(* Logix 5000 project; controller BreakGroup_US vendor 1 type 14 code 211 rev 32.16; software revision 32.05; part 3 of 8 *)
(* tags used below, declared in another part *)
   Emg_Stop : BOOL;
   Gantry_2_Horizontal_Start : BOOL;
   Gantry_2_Tilter_LH_Start : BOOL;
   Gantry_2_Tilter_RH_Start : BOOL;
   Gantry_2_vertical_Start : BOOL;
   HMI_Gantry_02_Hor_PB : SINT;
   HMI_Gantry_2_Tilter_LH_PB : SINT;
   HMI_Gantry_2_Tilter_RH_PB : SINT;
   HMI_Gantry_2_vertical_PB : SINT;
   HMI_MAN_GTY2_HORI_STOP : BOOL;
   HMI_MAN_GTY2_TIL2_STOP : BOOL;
   HMI_MAN_GTY2_VERT_STOP : BOOL;
   MAN_GTY2_HORI_HOME : TIMER;
   MAN_GTY2_TIL1_HOME : TIMER;
   MAN_GTY2_TIL2_HOME : TIMER;
   MAN_GTY2_VERT_HOME : TIMER;
   RCP_GY_02_Horizontal : RCP_Servo_02;
   RCP_GY_02_Vertical : RCP_Servo_02;
   RCP_Tilt_Axis_Master : RCP_Servo_02;
   RCP_Tilt_Axis_Slave : RCP_Servo_02;
   ST10_Trolley1Lock_Cyl_01_Extended : ALIAS FOR MCP_PT01:1:I.0;
   ST10_Trolley1LockCyl_01_Retracted : ALIAS FOR MCP_PT01:1:I.1;
   ST10_Trolley_Present_Sensor : ALIAS FOR MCP_PT01:1:I.2;
   ST10_TrolleyTopSideProductPresentSensor : ALIAS FOR MCP_PT01:1:I.3;
   ST20_Trolley_Present_Sensor_02 : ALIAS FOR MCP_PT01:1:I.6;
   ST20_TrolleyTopSideProductPresentSensor : ALIAS FOR MCP_PT01:4:I.3;
   ST30_Auto_SS : ALIAS FOR MCP_PT01:6:I.3;
   ST30_Emg_Push_Buttion : ALIAS FOR MCP_PT01:5:I.7;
   ST30_Home_PB : ALIAS FOR MCP_PT01:6:I.2;
   ST30_Hydro_motor : ALIAS FOR MCP_PT01:5:I.6;
   ST30_IndexingTableHomePositionSensor : ALIAS FOR MCP_PT01:4:I.5;
   ST30_IndexPlateLockCyl1Extended : ALIAS FOR MCP_PT01:4:I.6;
   ST30_IndexPlateLockCyl1Retracted : ALIAS FOR MCP_PT01:4:I.7;
   ST30_IndexPlateLockCyl2Extended : ALIAS FOR MCP_PT01:5:I.0;
   ST30_IndexPlateLockCyl2Retracted : ALIAS FOR MCP_PT01:5:I.1;
   ST30_Manual_SS : ALIAS FOR MCP_PT01:6:I.4;
   ST30_PressUnitCyl_1Extended : ALIAS FOR MCP_PT01:5:I.2;
   ST30_PressUnitCyl_1Retracted : ALIAS FOR MCP_PT01:5:I.3;
   ST30_PressUnitCyl_2Extended : ALIAS FOR MCP_PT01:5:I.4;
   ST30_PressUnitCyl_2Retracted : ALIAS FOR MCP_PT01:5:I.5;
   ST30_Product_Present_Sensor : ALIAS FOR MCP_PT01:4:I.4;
   ST30_Reset_PB : ALIAS FOR MCP_PT01:6:I.5;
   ST30_Start_PB : ALIAS FOR MCP_PT01:6:I.0;
   ST30_Stop_PB : ALIAS FOR MCP_PT01:6:I.1;
   ST40_Auto_SS : ALIAS FOR MCP_PT01:10:I.5;
   ST40_EMG_PB : ALIAS FOR MCP_PT01:10:I.1;
   ST40_Home_PB : ALIAS FOR MCP_PT01:10:I.4;
   ST40_IndexingTableHomePositionSensor : ALIAS FOR MCP_PT01:6:I.7;
   ST40_IndexPlateLockCyl01_Extended : ALIAS FOR MCP_PT01:7:I.0;
   ST40_IndexPlateLockCyl01_Retracted : ALIAS FOR MCP_PT01:7:I.1;
   ST40_IndexPlateLockCyl02_Extended : ALIAS FOR MCP_PT01:7:I.2;
   ST40_IndexPlateLockCyl02_Retracted : ALIAS FOR MCP_PT01:7:I.3;
   ST40_Manual_SS : ALIAS FOR MCP_PT01:10:I.6;
   ST40_ProductPresentSensor : ALIAS FOR MCP_PT01:6:I.6;
   ST40_Reset_PB : ALIAS FOR MCP_PT01:10:I.7;
   ST40_Start_PB : ALIAS FOR MCP_PT01:10:I.2;
   ST40_Stop_PB : ALIAS FOR MCP_PT01:10:I.3;
   ST50_Auto_SS : ALIAS FOR MCP_PT01:15:I.1;
   ST50_Conv_End_Sensor : ALIAS FOR MCP_PT01:11:I.7;
   ST50_Conv_Home_Sensor : ALIAS FOR MCP_PT01:11:I.6;
   ST50_EMG_PB : ALIAS FOR MCP_PT01:14:I.5;
   ST50_Home_PB : ALIAS FOR MCP_PT01:15:I.0;
   ST50_IndexPlateLockCyl01_Extended : ALIAS FOR MCP_PT01:11:I.2;
   ST50_IndexPlateLockCyl01_Retracted : ALIAS FOR MCP_PT01:11:I.3;
   ST50_IndexPlateLockCyl02_Extended : ALIAS FOR MCP_PT01:11:I.4;
   ST50_IndexPlateLockCyl02_Retracted : ALIAS FOR MCP_PT01:11:I.5;
   ST50_IndexTableHomePositionSensor : ALIAS FOR MCP_PT01:11:I.1;
   ST50_Manual_SS : ALIAS FOR MCP_PT01:15:I.2;
   ST50_Product_Present_Sensor : ALIAS FOR MCP_PT01:11:I.0;
   ST50_Reset_PB : ALIAS FOR MCP_PT01:15:I.3;
   ST50_Start_PB : ALIAS FOR MCP_PT01:14:I.6;
   ST50_Stop_PB : ALIAS FOR MCP_PT01:14:I.7;
   ST60_Auto_SS : ALIAS FOR MCP_PT01:20:I.2;
   ST60_Conv_End_Sensor : ALIAS FOR MCP_PT01:16:I.3;
   ST60_Conv_Home_Sensor : ALIAS FOR MCP_PT01:16:I.2;
   ST60_EMG_PB : ALIAS FOR MCP_PT01:19:I.6;
   ST60_Home_PB : ALIAS FOR MCP_PT01:20:I.1;
   ST60_Hydro_Motor : ALIAS FOR MCP_PT01:17:I.0;
   ST60_IndexPlateLockCyl01_Extended : ALIAS FOR MCP_PT01:15:I.6;
   ST60_IndexPlateLockCyl01_Retracted : ALIAS FOR MCP_PT01:15:I.7;
   ST60_IndexPlateLockCyl02_Extended : ALIAS FOR MCP_PT01:16:I.0;
   ST60_IndexPlateLockCyl02_Retracted : ALIAS FOR MCP_PT01:16:I.1;
   ST60_IndexTableHomePositionSensor : ALIAS FOR MCP_PT01:15:I.5;
   ST60_Manual_SS : ALIAS FOR MCP_PT01:20:I.3;
   ST60_Press_Unit_Cyl01_Extended : ALIAS FOR MCP_PT01:16:I.4;
   ST60_Press_Unit_Cyl01_Retracted : ALIAS FOR MCP_PT01:16:I.5;
   ST60_Press_Unit_Cyl02_Extended : ALIAS FOR MCP_PT01:16:I.6;
   ST60_Press_Unit_Cyl02_Retracted : ALIAS FOR MCP_PT01:16:I.7;
   ST60_Product_Present_Sensor : ALIAS FOR MCP_PT01:15:I.4;
   ST60_Reset_PB : ALIAS FOR MCP_PT01:20:I.4;
   ST60_Start_PB : ALIAS FOR MCP_PT01:19:I.7;
   ST60_Stop_PB : ALIAS FOR MCP_PT01:20:I.0;
   ST70_Auto_SS : ALIAS FOR MCP_PT01:22:I.1;
   ST70_Conv_End_Sensor : ALIAS FOR MCP_PT01:21:I.4;
   ST70_Conv_Home_Sensor : ALIAS FOR MCP_PT01:21:I.3;
   ST70_EMG_PB : ALIAS FOR MCP_PT01:21:I.5;
   ST70_Home_PB : ALIAS FOR MCP_PT01:22:I.0;
   ST70_IndexPlateLockCyl01_Extended : ALIAS FOR MCP_PT01:20:I.7;
   ST70_IndexPlateLockCyl01_Retracted : ALIAS FOR MCP_PT01:21:I.0;
   ST70_IndexPlateLockCyl02_Extended : ALIAS FOR MCP_PT01:21:I.1;
   ST70_IndexPlateLockCyl02_Retracted : ALIAS FOR MCP_PT01:21:I.2;
   ST70_IndexTableHomePositionSensor : ALIAS FOR MCP_PT01:20:I.6;
   ST70_Manual_SS : ALIAS FOR MCP_PT01:22:I.2;
   ST70_Product_Present_Sensor : ALIAS FOR MCP_PT01:20:I.5;
   ST70_Reset_PB : ALIAS FOR MCP_PT01:22:I.3;
   ST70_Start_PB : ALIAS FOR MCP_PT01:21:I.6;
   ST70_Stop_PB : ALIAS FOR MCP_PT01:21:I.7;
   ST_20Trolley_1LockCylExtended : ALIAS FOR MCP_PT01:1:I.4;
   ST_20Trolley_1LockingCylRetracted : ALIAS FOR MCP_PT01:1:I.5;
   TEST_02 : BOOL;

PROGRAM Gantry_02_Horizontal   (* main routine Main *)

ROUTINE Main   (* ladder *)
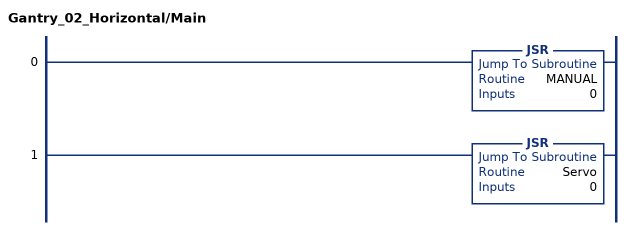
   0: JSR(MANUAL,0);
   1: JSR(Servo,0);
END_ROUTINE

ROUTINE MANUAL   (* ladder *)
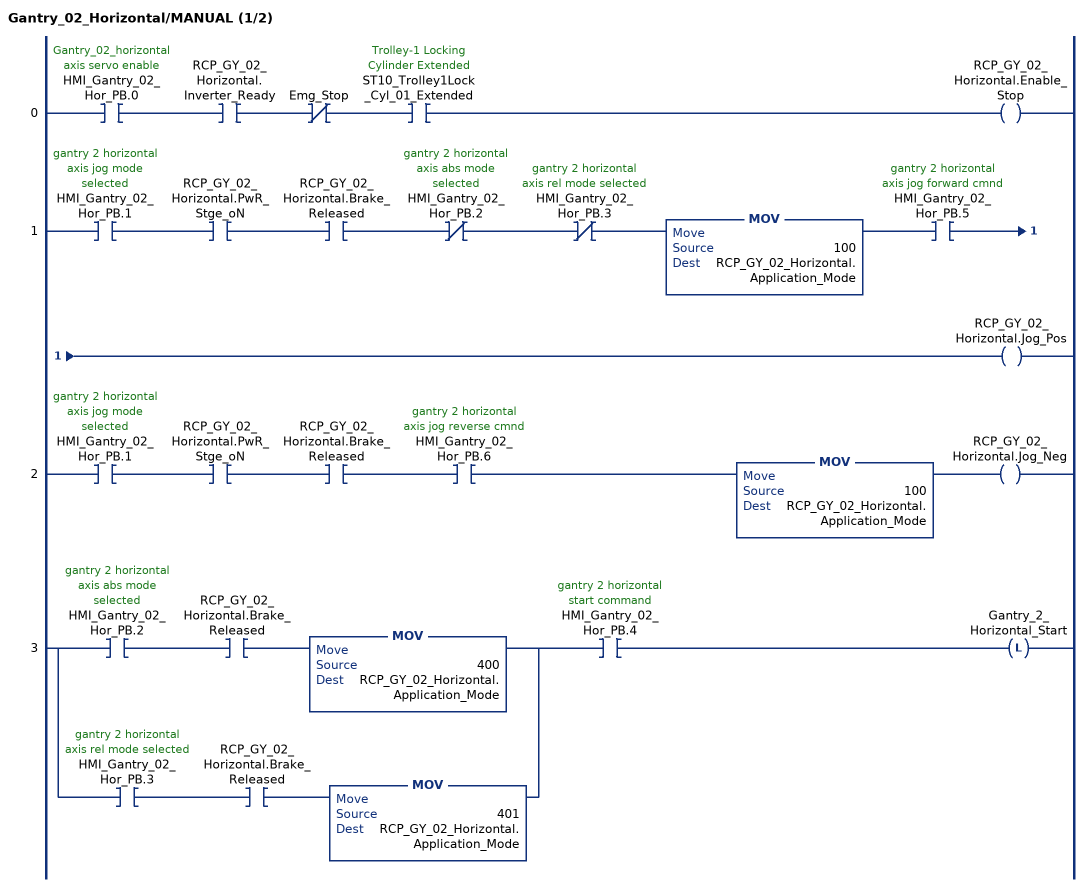
   0: XIC(HMI_Gantry_02_Hor_PB.0)XIC(RCP_GY_02_Horizontal.Inverter_Ready)XIO(Emg_Stop)XIC(ST10_Trolley1Lock_Cyl_01_Extended)OTE(RCP_GY_02_Horizontal.Enable_Stop);
   1: XIC(HMI_Gantry_02_Hor_PB.1)XIC(RCP_GY_02_Horizontal.PwR_Stge_oN)XIC(RCP_GY_02_Horizontal.Brake_Released)XIO(HMI_Gantry_02_Hor_PB.2)XIO(HMI_Gantry_02_Hor_PB.3)MOV(100,RCP_GY_02_Horizontal.Application_Mode)XIC(HMI_Gantry_02_Hor_PB.5)OTE(RCP_GY_02_Horizontal.Jog_Pos);
   2: XIC(HMI_Gantry_02_Hor_PB.1)XIC(RCP_GY_02_Horizontal.PwR_Stge_oN)XIC(RCP_GY_02_Horizontal.Brake_Released)XIC(HMI_Gantry_02_Hor_PB.6)MOV(100,RCP_GY_02_Horizontal.Application_Mode)OTE(RCP_GY_02_Horizontal.Jog_Neg);
   3: [XIC(HMI_Gantry_02_Hor_PB.2) XIC(RCP_GY_02_Horizontal.Brake_Released) MOV(400,RCP_GY_02_Horizontal.Application_Mode) ,XIC(HMI_Gantry_02_Hor_PB.3) XIC(RCP_GY_02_Horizontal.Brake_Released) MOV(401,RCP_GY_02_Horizontal.Application_Mode) ]XIC(HMI_Gantry_02_Hor_PB.4)OTL(Gantry_2_Horizontal_Start);
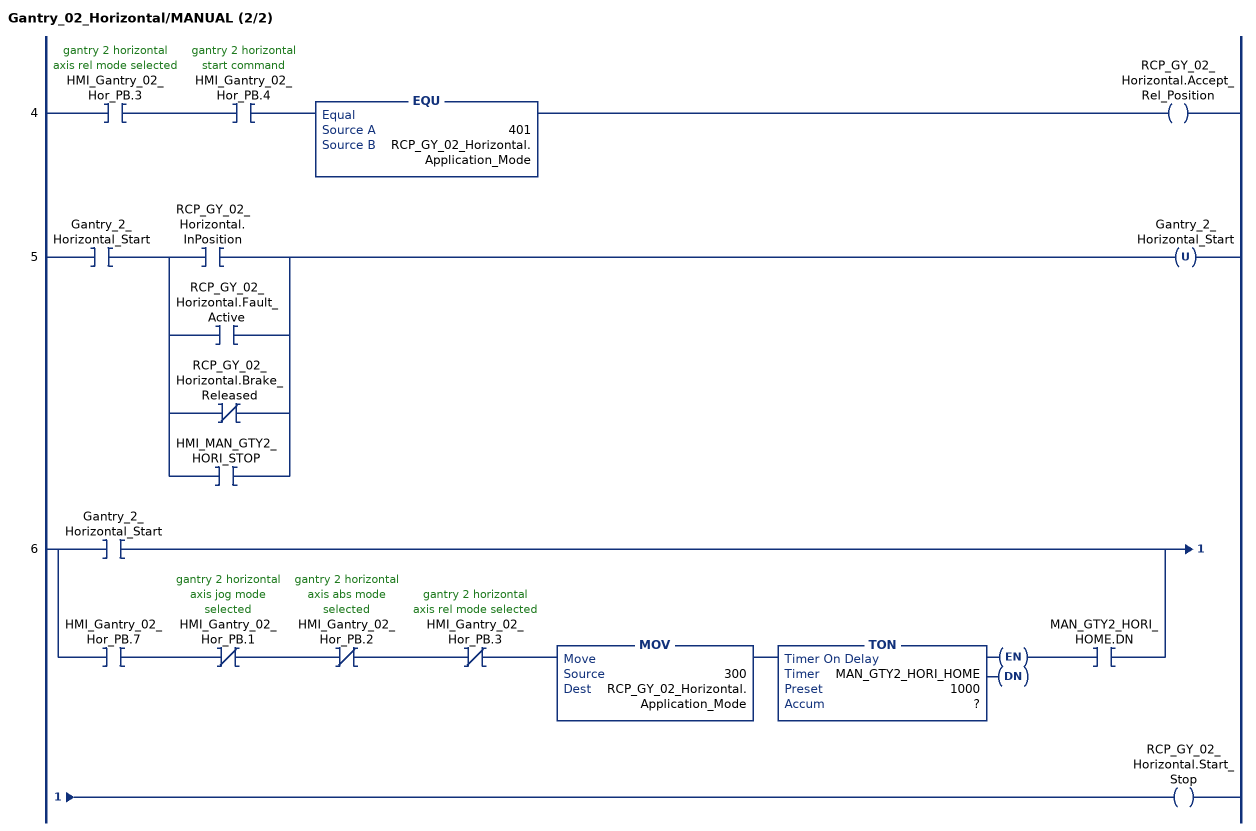
   4: XIC(HMI_Gantry_02_Hor_PB.3)XIC(HMI_Gantry_02_Hor_PB.4)EQU(401,RCP_GY_02_Horizontal.Application_Mode)OTE(RCP_GY_02_Horizontal.Accept_Rel_Position);
   5: XIC(Gantry_2_Horizontal_Start)[XIC(RCP_GY_02_Horizontal.InPosition) ,[XIC(RCP_GY_02_Horizontal.Fault_Active) ,[XIO(RCP_GY_02_Horizontal.Brake_Released) ,XIC(HMI_MAN_GTY2_HORI_STOP) ] ] ]OTU(Gantry_2_Horizontal_Start);
   6: [XIC(Gantry_2_Horizontal_Start) ,XIC(HMI_Gantry_02_Hor_PB.7) XIO(HMI_Gantry_02_Hor_PB.1) XIO(HMI_Gantry_02_Hor_PB.2) XIO(HMI_Gantry_02_Hor_PB.3) MOV(300,RCP_GY_02_Horizontal.Application_Mode) TON(MAN_GTY2_HORI_HOME,?,?) XIC(MAN_GTY2_HORI_HOME.DN) ]OTE(RCP_GY_02_Horizontal.Start_Stop);
END_ROUTINE

ROUTINE Servo   (* ladder *)
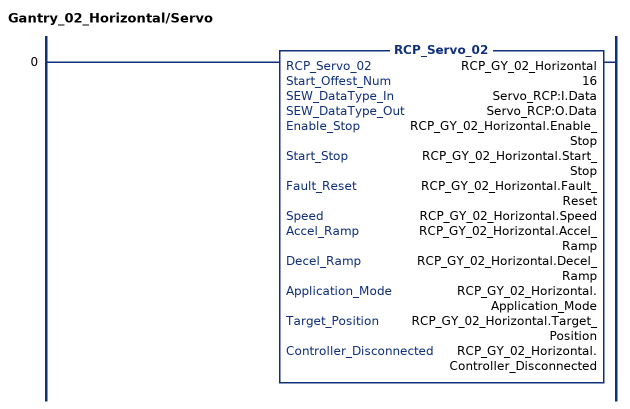
   0: RCP_Servo_02(RCP_GY_02_Horizontal,16,Servo_RCP:I.Data,Servo_RCP:O.Data,RCP_GY_02_Horizontal.Enable_Stop,RCP_GY_02_Horizontal.Start_Stop,RCP_GY_02_Horizontal.Fault_Reset,RCP_GY_02_Horizontal.Speed,RCP_GY_02_Horizontal.Accel_Ramp,RCP_GY_02_Horizontal.Decel_Ramp,RCP_GY_02_Horizontal.Application_Mode,RCP_GY_02_Horizontal.Target_Position,RCP_GY_02_Horizontal.Controller_Disconnected);
END_ROUTINE
END_PROGRAM

PROGRAM Gantry_02_Tilter   (* main routine Main *)

ROUTINE Main   (* ladder *)
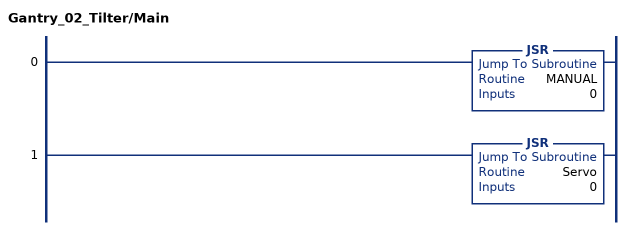
   0: JSR(MANUAL,0);
   1: JSR(Servo,0);
END_ROUTINE

ROUTINE MANUAL   (* ladder *)
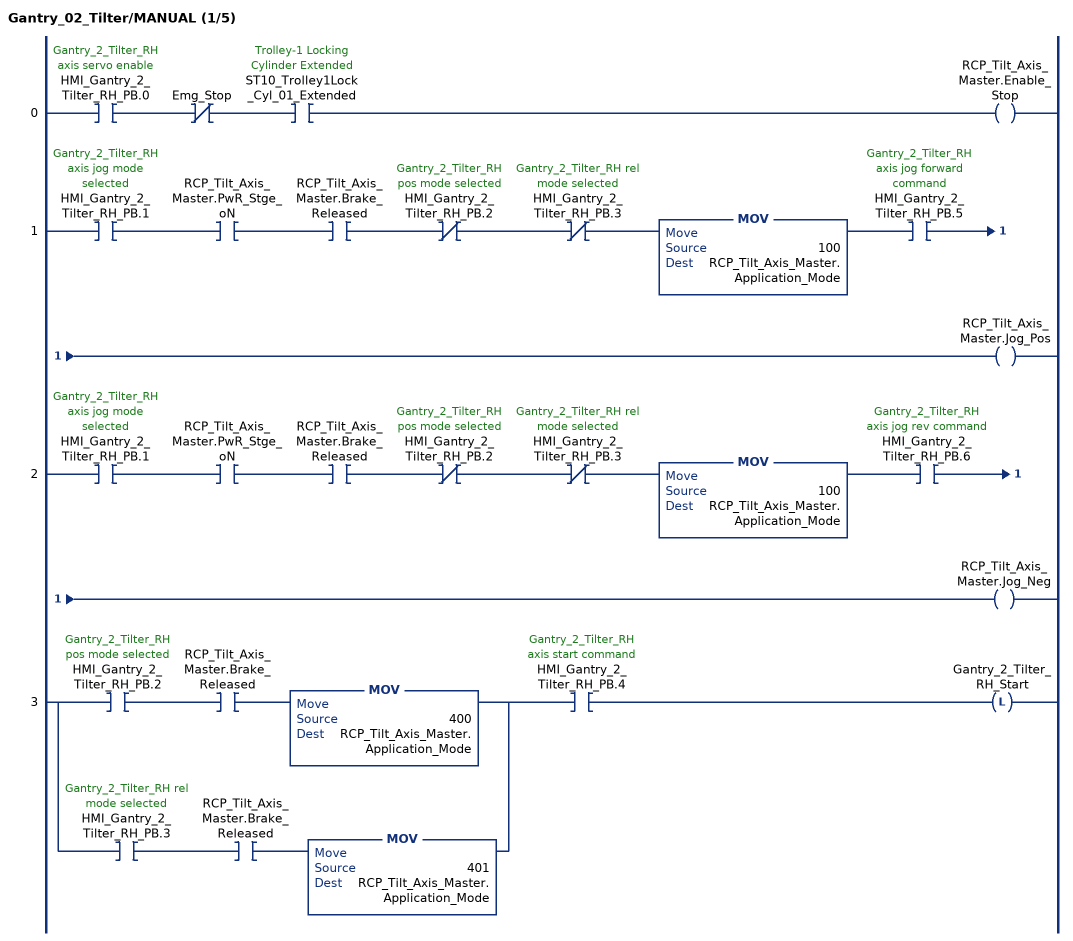
   0: XIC(HMI_Gantry_2_Tilter_RH_PB.0)XIO(Emg_Stop)XIC(ST10_Trolley1Lock_Cyl_01_Extended)OTE(RCP_Tilt_Axis_Master.Enable_Stop);
   1: XIC(HMI_Gantry_2_Tilter_RH_PB.1)XIC(RCP_Tilt_Axis_Master.PwR_Stge_oN)XIC(RCP_Tilt_Axis_Master.Brake_Released)XIO(HMI_Gantry_2_Tilter_RH_PB.2)XIO(HMI_Gantry_2_Tilter_RH_PB.3)MOV(100,RCP_Tilt_Axis_Master.Application_Mode)XIC(HMI_Gantry_2_Tilter_RH_PB.5)OTE(RCP_Tilt_Axis_Master.Jog_Pos);
   2: XIC(HMI_Gantry_2_Tilter_RH_PB.1)XIC(RCP_Tilt_Axis_Master.PwR_Stge_oN)XIC(RCP_Tilt_Axis_Master.Brake_Released)XIO(HMI_Gantry_2_Tilter_RH_PB.2)XIO(HMI_Gantry_2_Tilter_RH_PB.3)MOV(100,RCP_Tilt_Axis_Master.Application_Mode)XIC(HMI_Gantry_2_Tilter_RH_PB.6)OTE(RCP_Tilt_Axis_Master.Jog_Neg);
   3: [XIC(HMI_Gantry_2_Tilter_RH_PB.2) XIC(RCP_Tilt_Axis_Master.Brake_Released) MOV(400,RCP_Tilt_Axis_Master.Application_Mode) ,XIC(HMI_Gantry_2_Tilter_RH_PB.3) XIC(RCP_Tilt_Axis_Master.Brake_Released) MOV(401,RCP_Tilt_Axis_Master.Application_Mode) ]XIC(HMI_Gantry_2_Tilter_RH_PB.4)OTL(Gantry_2_Tilter_RH_Start);
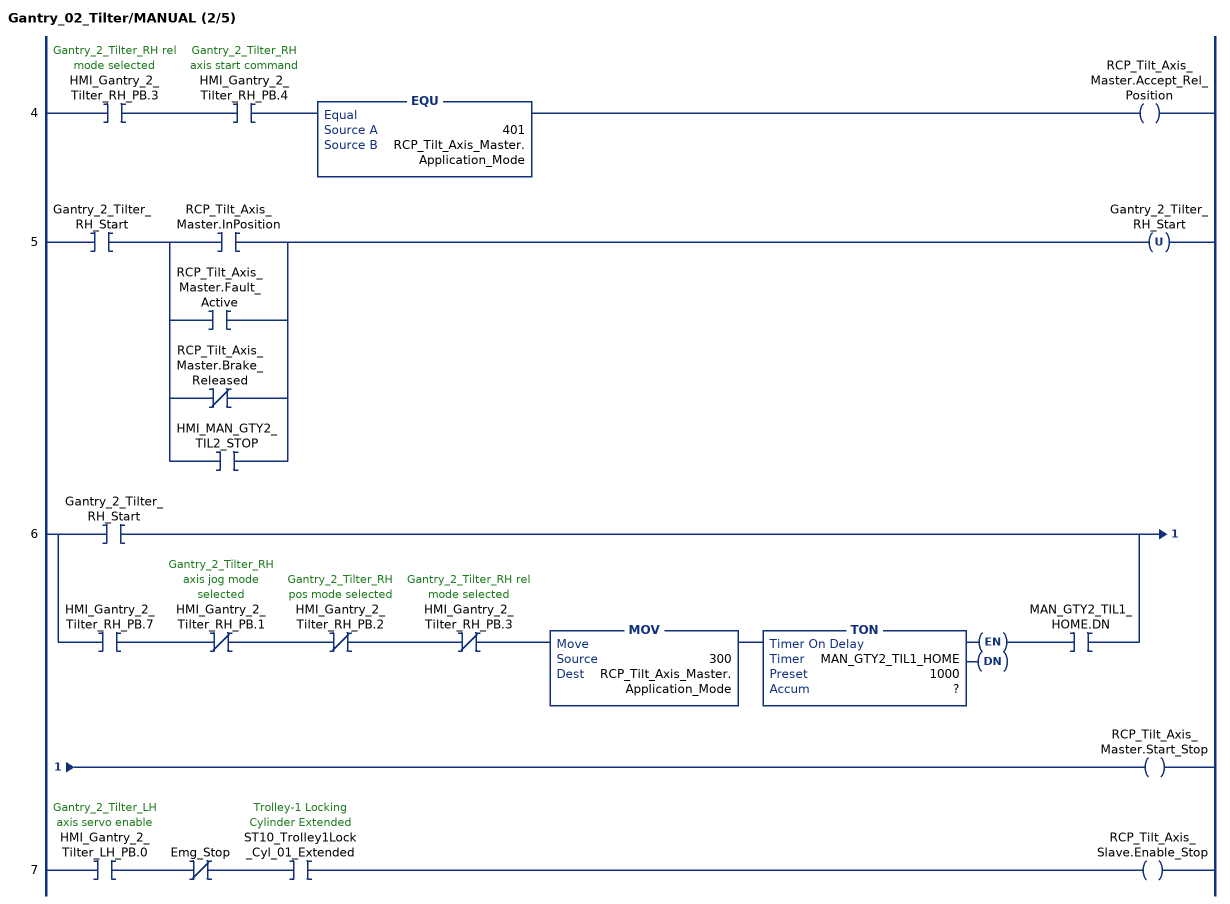
   4: XIC(HMI_Gantry_2_Tilter_RH_PB.3)XIC(HMI_Gantry_2_Tilter_RH_PB.4)EQU(401,RCP_Tilt_Axis_Master.Application_Mode)OTE(RCP_Tilt_Axis_Master.Accept_Rel_Position);
   5: XIC(Gantry_2_Tilter_RH_Start)[XIC(RCP_Tilt_Axis_Master.InPosition) ,[XIC(RCP_Tilt_Axis_Master.Fault_Active) ,[XIO(RCP_Tilt_Axis_Master.Brake_Released) ,XIC(HMI_MAN_GTY2_TIL2_STOP) ] ] ]OTU(Gantry_2_Tilter_RH_Start);
   6: [XIC(Gantry_2_Tilter_RH_Start) ,XIC(HMI_Gantry_2_Tilter_RH_PB.7) XIO(HMI_Gantry_2_Tilter_RH_PB.1) XIO(HMI_Gantry_2_Tilter_RH_PB.2) XIO(HMI_Gantry_2_Tilter_RH_PB.3) MOV(300,RCP_Tilt_Axis_Master.Application_Mode) TON(MAN_GTY2_TIL1_HOME,?,?) XIC(MAN_GTY2_TIL1_HOME.DN) ]OTE(RCP_Tilt_Axis_Master.Start_Stop);
   7: XIC(HMI_Gantry_2_Tilter_LH_PB.0)XIO(Emg_Stop)XIC(ST10_Trolley1Lock_Cyl_01_Extended)OTE(RCP_Tilt_Axis_Slave.Enable_Stop);
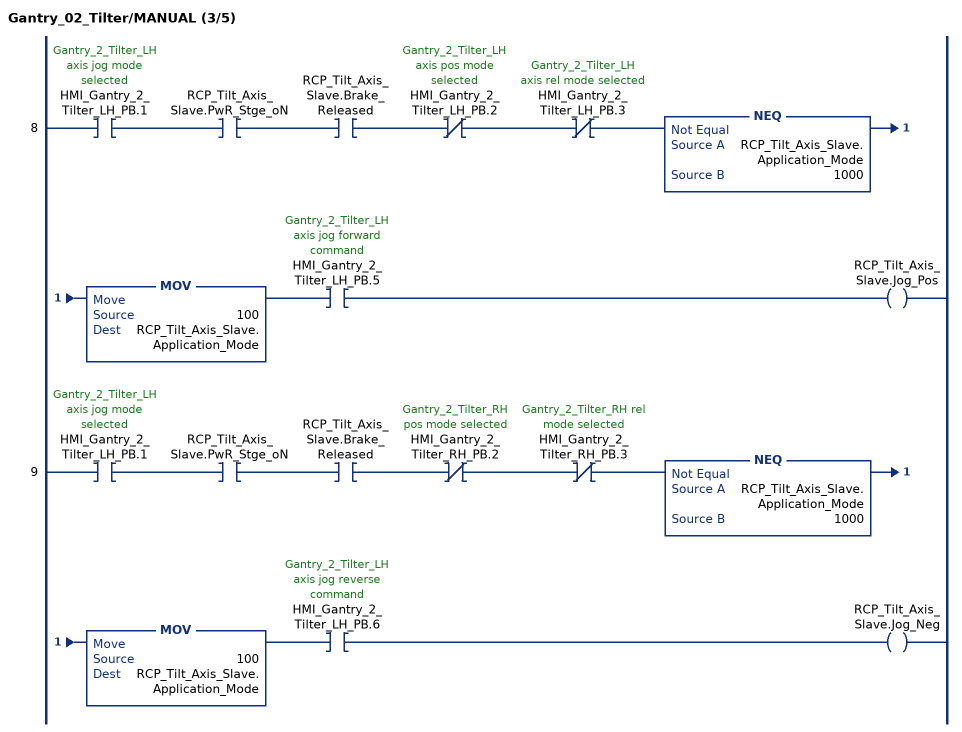
   8: XIC(HMI_Gantry_2_Tilter_LH_PB.1)XIC(RCP_Tilt_Axis_Slave.PwR_Stge_oN)XIC(RCP_Tilt_Axis_Slave.Brake_Released)XIO(HMI_Gantry_2_Tilter_LH_PB.2)XIO(HMI_Gantry_2_Tilter_LH_PB.3)NEQ(RCP_Tilt_Axis_Slave.Application_Mode,1000)MOV(100,RCP_Tilt_Axis_Slave.Application_Mode)XIC(HMI_Gantry_2_Tilter_LH_PB.5)OTE(RCP_Tilt_Axis_Slave.Jog_Pos);
   9: XIC(HMI_Gantry_2_Tilter_LH_PB.1)XIC(RCP_Tilt_Axis_Slave.PwR_Stge_oN)XIC(RCP_Tilt_Axis_Slave.Brake_Released)XIO(HMI_Gantry_2_Tilter_RH_PB.2)XIO(HMI_Gantry_2_Tilter_RH_PB.3)NEQ(RCP_Tilt_Axis_Slave.Application_Mode,1000)MOV(100,RCP_Tilt_Axis_Slave.Application_Mode)XIC(HMI_Gantry_2_Tilter_LH_PB.6)OTE(RCP_Tilt_Axis_Slave.Jog_Neg);
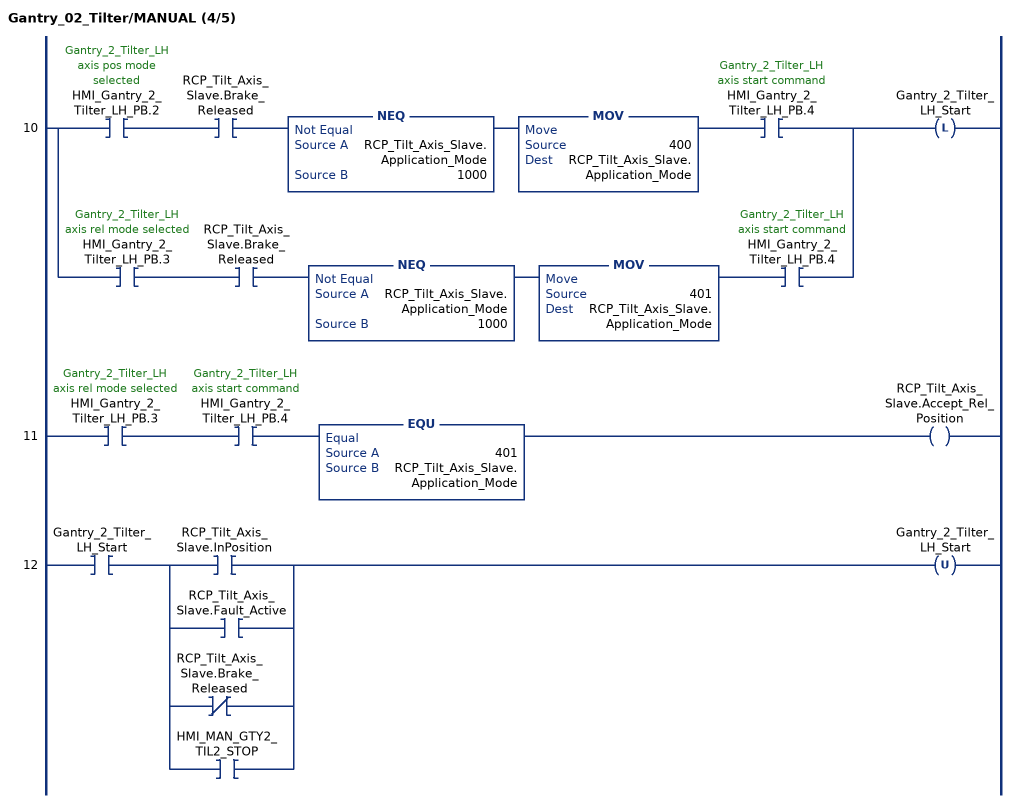
   10: [XIC(HMI_Gantry_2_Tilter_LH_PB.2) XIC(RCP_Tilt_Axis_Slave.Brake_Released) NEQ(RCP_Tilt_Axis_Slave.Application_Mode,1000) MOV(400,RCP_Tilt_Axis_Slave.Application_Mode) XIC(HMI_Gantry_2_Tilter_LH_PB.4) ,XIC(HMI_Gantry_2_Tilter_LH_PB.3) XIC(RCP_Tilt_Axis_Slave.Brake_Released) NEQ(RCP_Tilt_Axis_Slave.Application_Mode,1000) MOV(401,RCP_Tilt_Axis_Slave.Application_Mode) XIC(HMI_Gantry_2_Tilter_LH_PB.4) ]OTL(Gantry_2_Tilter_LH_Start);
   11: XIC(HMI_Gantry_2_Tilter_LH_PB.3)XIC(HMI_Gantry_2_Tilter_LH_PB.4)EQU(401,RCP_Tilt_Axis_Slave.Application_Mode)OTE(RCP_Tilt_Axis_Slave.Accept_Rel_Position);
   12: XIC(Gantry_2_Tilter_LH_Start)[XIC(RCP_Tilt_Axis_Slave.InPosition) ,[XIC(RCP_Tilt_Axis_Slave.Fault_Active) ,[XIO(RCP_Tilt_Axis_Slave.Brake_Released) ,XIC(HMI_MAN_GTY2_TIL2_STOP) ] ] ]OTU(Gantry_2_Tilter_LH_Start);
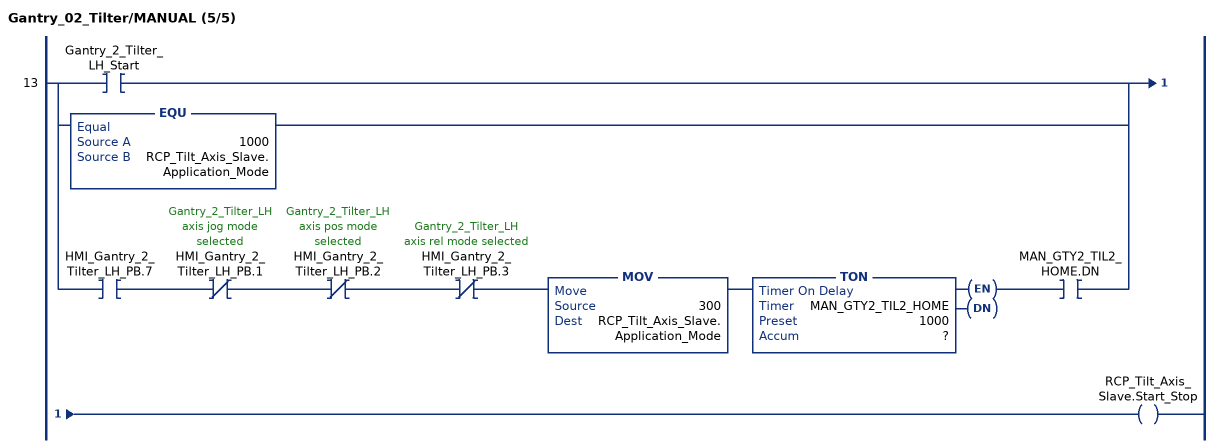
   13: [[XIC(Gantry_2_Tilter_LH_Start) ,EQU(1000,RCP_Tilt_Axis_Slave.Application_Mode) ] ,XIC(HMI_Gantry_2_Tilter_LH_PB.7) XIO(HMI_Gantry_2_Tilter_LH_PB.1) XIO(HMI_Gantry_2_Tilter_LH_PB.2) XIO(HMI_Gantry_2_Tilter_LH_PB.3) MOV(300,RCP_Tilt_Axis_Slave.Application_Mode) TON(MAN_GTY2_TIL2_HOME,?,?) XIC(MAN_GTY2_TIL2_HOME.DN) ]OTE(RCP_Tilt_Axis_Slave.Start_Stop);
END_ROUTINE

ROUTINE Servo   (* ladder *)
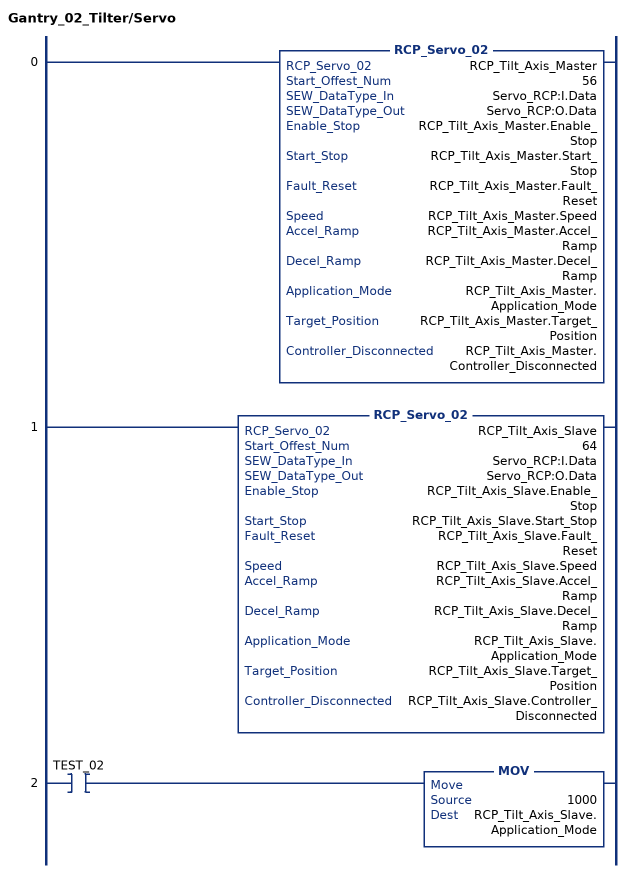
   0: RCP_Servo_02(RCP_Tilt_Axis_Master,56,Servo_RCP:I.Data,Servo_RCP:O.Data,RCP_Tilt_Axis_Master.Enable_Stop,RCP_Tilt_Axis_Master.Start_Stop,RCP_Tilt_Axis_Master.Fault_Reset,RCP_Tilt_Axis_Master.Speed,RCP_Tilt_Axis_Master.Accel_Ramp,RCP_Tilt_Axis_Master.Decel_Ramp,RCP_Tilt_Axis_Master.Application_Mode,RCP_Tilt_Axis_Master.Target_Position,RCP_Tilt_Axis_Master.Controller_Disconnected);
   1: RCP_Servo_02(RCP_Tilt_Axis_Slave,64,Servo_RCP:I.Data,Servo_RCP:O.Data,RCP_Tilt_Axis_Slave.Enable_Stop,RCP_Tilt_Axis_Slave.Start_Stop,RCP_Tilt_Axis_Slave.Fault_Reset,RCP_Tilt_Axis_Slave.Speed,RCP_Tilt_Axis_Slave.Accel_Ramp,RCP_Tilt_Axis_Slave.Decel_Ramp,RCP_Tilt_Axis_Slave.Application_Mode,RCP_Tilt_Axis_Slave.Target_Position,RCP_Tilt_Axis_Slave.Controller_Disconnected);
   2: XIC(TEST_02)MOV(1000,RCP_Tilt_Axis_Slave.Application_Mode);
END_ROUTINE
END_PROGRAM

PROGRAM Gantry_02_Vertical   (* main routine Main *)

ROUTINE Main   (* ladder *)
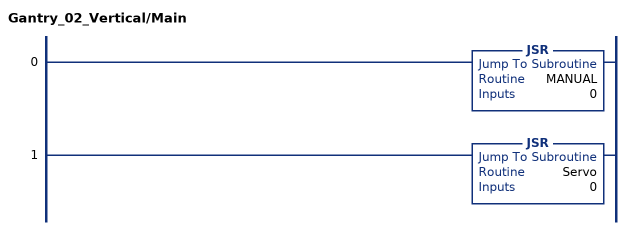
   0: JSR(MANUAL,0);
   1: JSR(Servo,0);
END_ROUTINE

ROUTINE MANUAL   (* ladder *)
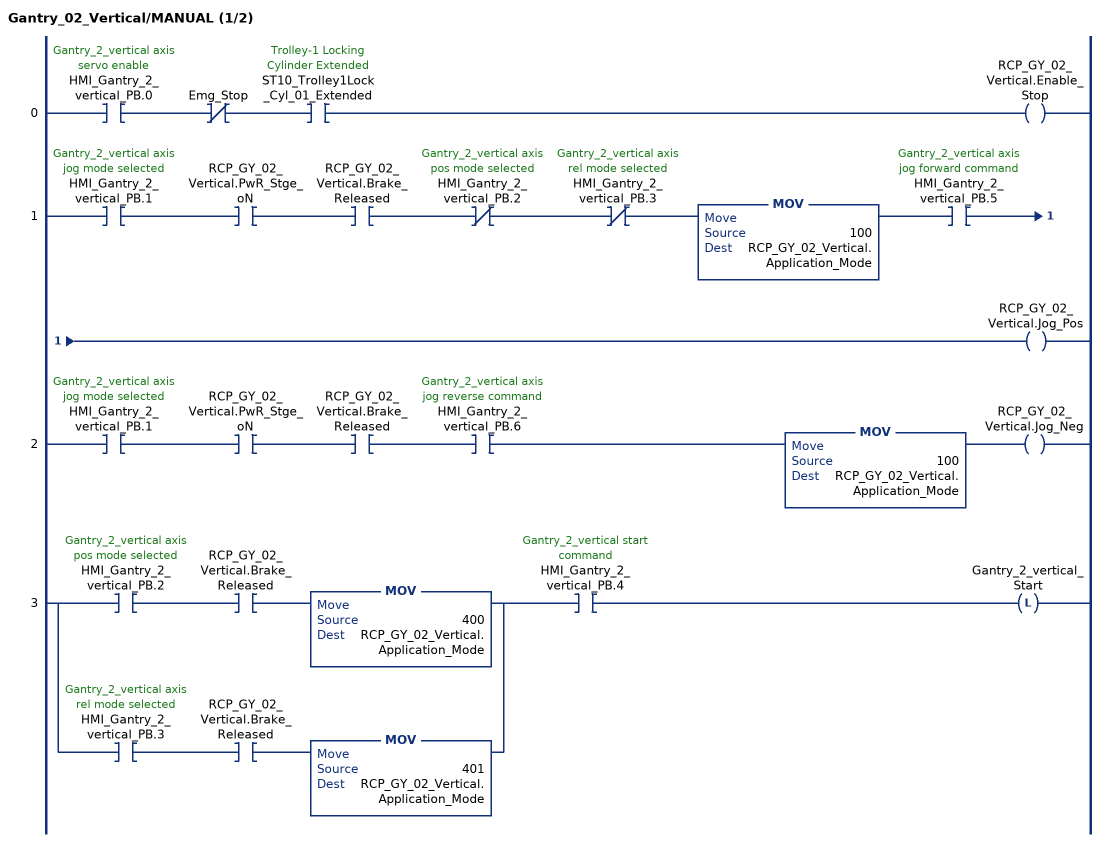
   0: XIC(HMI_Gantry_2_vertical_PB.0)XIO(Emg_Stop)XIC(ST10_Trolley1Lock_Cyl_01_Extended)OTE(RCP_GY_02_Vertical.Enable_Stop);
   1: XIC(HMI_Gantry_2_vertical_PB.1)XIC(RCP_GY_02_Vertical.PwR_Stge_oN)XIC(RCP_GY_02_Vertical.Brake_Released)XIO(HMI_Gantry_2_vertical_PB.2)XIO(HMI_Gantry_2_vertical_PB.3)MOV(100,RCP_GY_02_Vertical.Application_Mode)XIC(HMI_Gantry_2_vertical_PB.5)OTE(RCP_GY_02_Vertical.Jog_Pos);
   2: XIC(HMI_Gantry_2_vertical_PB.1)XIC(RCP_GY_02_Vertical.PwR_Stge_oN)XIC(RCP_GY_02_Vertical.Brake_Released)XIC(HMI_Gantry_2_vertical_PB.6)MOV(100,RCP_GY_02_Vertical.Application_Mode)OTE(RCP_GY_02_Vertical.Jog_Neg);
   3: [XIC(HMI_Gantry_2_vertical_PB.2) XIC(RCP_GY_02_Vertical.Brake_Released) MOV(400,RCP_GY_02_Vertical.Application_Mode) ,XIC(HMI_Gantry_2_vertical_PB.3) XIC(RCP_GY_02_Vertical.Brake_Released) MOV(401,RCP_GY_02_Vertical.Application_Mode) ]XIC(HMI_Gantry_2_vertical_PB.4)OTL(Gantry_2_vertical_Start);
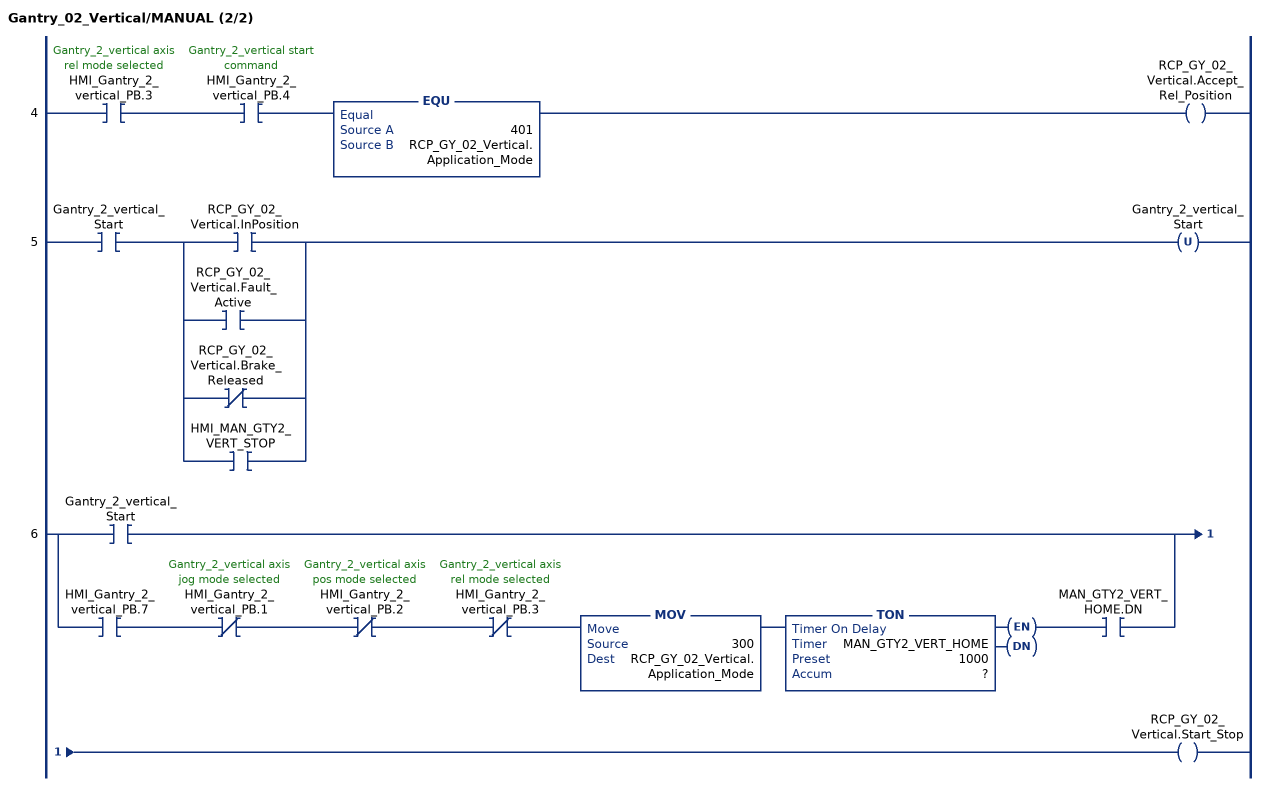
   4: XIC(HMI_Gantry_2_vertical_PB.3)XIC(HMI_Gantry_2_vertical_PB.4)EQU(401,RCP_GY_02_Vertical.Application_Mode)OTE(RCP_GY_02_Vertical.Accept_Rel_Position);
   5: XIC(Gantry_2_vertical_Start)[XIC(RCP_GY_02_Vertical.InPosition) ,[XIC(RCP_GY_02_Vertical.Fault_Active) ,[XIO(RCP_GY_02_Vertical.Brake_Released) ,XIC(HMI_MAN_GTY2_VERT_STOP) ] ] ]OTU(Gantry_2_vertical_Start);
   6: [XIC(Gantry_2_vertical_Start) ,XIC(HMI_Gantry_2_vertical_PB.7) XIO(HMI_Gantry_2_vertical_PB.1) XIO(HMI_Gantry_2_vertical_PB.2) XIO(HMI_Gantry_2_vertical_PB.3) MOV(300,RCP_GY_02_Vertical.Application_Mode) TON(MAN_GTY2_VERT_HOME,?,?) XIC(MAN_GTY2_VERT_HOME.DN) ]OTE(RCP_GY_02_Vertical.Start_Stop);
END_ROUTINE

ROUTINE Servo   (* ladder *)
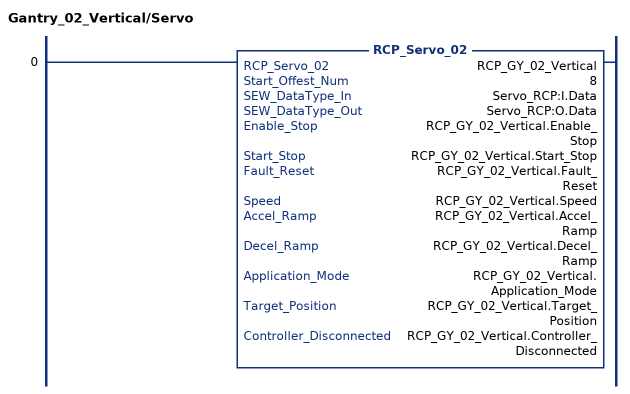
   0: RCP_Servo_02(RCP_GY_02_Vertical,8,Servo_RCP:I.Data,Servo_RCP:O.Data,RCP_GY_02_Vertical.Enable_Stop,RCP_GY_02_Vertical.Start_Stop,RCP_GY_02_Vertical.Fault_Reset,RCP_GY_02_Vertical.Speed,RCP_GY_02_Vertical.Accel_Ramp,RCP_GY_02_Vertical.Decel_Ramp,RCP_GY_02_Vertical.Application_Mode,RCP_GY_02_Vertical.Target_Position,RCP_GY_02_Vertical.Controller_Disconnected);
END_ROUTINE
END_PROGRAM

PROGRAM MainProgram   (* main routine Main *)

ROUTINE IP_Map   (* ladder *)
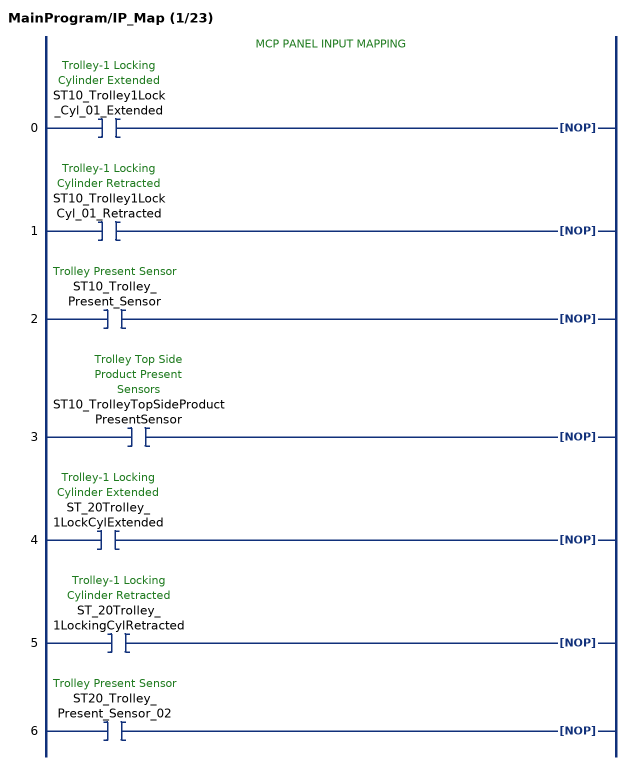
   // MCP PANEL INPUT MAPPING
   0: XIC(ST10_Trolley1Lock_Cyl_01_Extended)NOP();
   1: XIC(ST10_Trolley1LockCyl_01_Retracted)NOP();
   2: XIC(ST10_Trolley_Present_Sensor)NOP();
   3: XIC(ST10_TrolleyTopSideProductPresentSensor)NOP();
   4: XIC(ST_20Trolley_1LockCylExtended)NOP();
   5: XIC(ST_20Trolley_1LockingCylRetracted)NOP();
   6: XIC(ST20_Trolley_Present_Sensor_02)NOP();
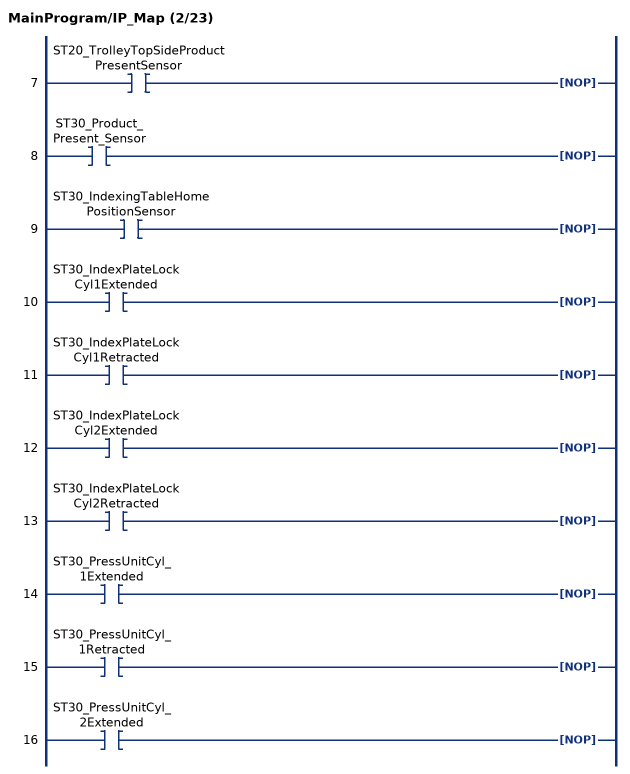
   7: XIC(ST20_TrolleyTopSideProductPresentSensor)NOP();
   8: XIC(ST30_Product_Present_Sensor)NOP();
   9: XIC(ST30_IndexingTableHomePositionSensor)NOP();
   10: XIC(ST30_IndexPlateLockCyl1Extended)NOP();
   11: XIC(ST30_IndexPlateLockCyl1Retracted)NOP();
   12: XIC(ST30_IndexPlateLockCyl2Extended)NOP();
   13: XIC(ST30_IndexPlateLockCyl2Retracted)NOP();
   14: XIC(ST30_PressUnitCyl_1Extended)NOP();
   15: XIC(ST30_PressUnitCyl_1Retracted)NOP();
   16: XIC(ST30_PressUnitCyl_2Extended)NOP();
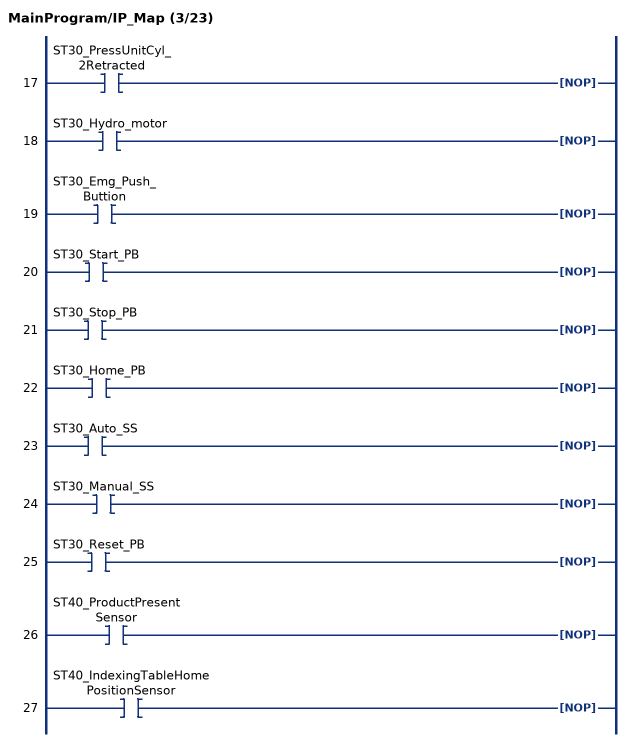
   17: XIC(ST30_PressUnitCyl_2Retracted)NOP();
   18: XIC(ST30_Hydro_motor)NOP();
   19: XIC(ST30_Emg_Push_Buttion)NOP();
   20: XIC(ST30_Start_PB)NOP();
   21: XIC(ST30_Stop_PB)NOP();
   22: XIC(ST30_Home_PB)NOP();
   23: XIC(ST30_Auto_SS)NOP();
   24: XIC(ST30_Manual_SS)NOP();
   25: XIC(ST30_Reset_PB)NOP();
   26: XIC(ST40_ProductPresentSensor)NOP();
   27: XIC(ST40_IndexingTableHomePositionSensor)NOP();
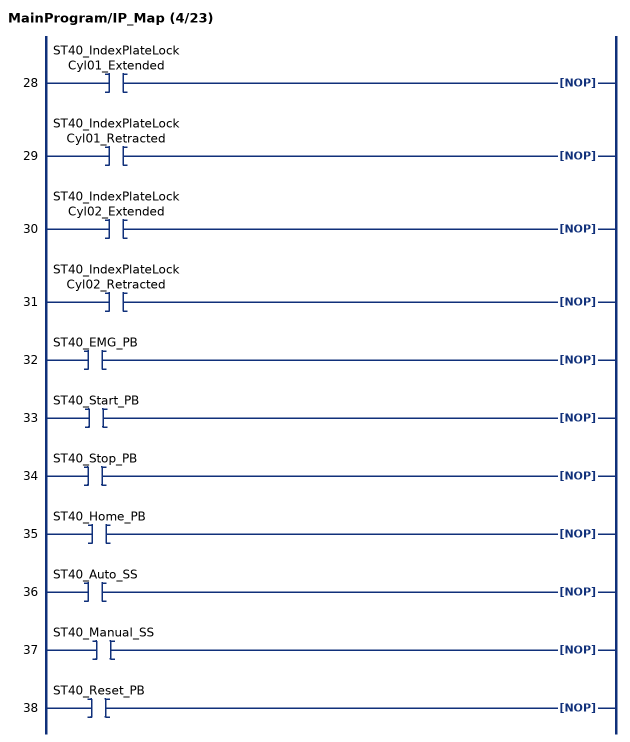
   28: XIC(ST40_IndexPlateLockCyl01_Extended)NOP();
   29: XIC(ST40_IndexPlateLockCyl01_Retracted)NOP();
   30: XIC(ST40_IndexPlateLockCyl02_Extended)NOP();
   31: XIC(ST40_IndexPlateLockCyl02_Retracted)NOP();
   32: XIC(ST40_EMG_PB)NOP();
   33: XIC(ST40_Start_PB)NOP();
   34: XIC(ST40_Stop_PB)NOP();
   35: XIC(ST40_Home_PB)NOP();
   36: XIC(ST40_Auto_SS)NOP();
   37: XIC(ST40_Manual_SS)NOP();
   38: XIC(ST40_Reset_PB)NOP();
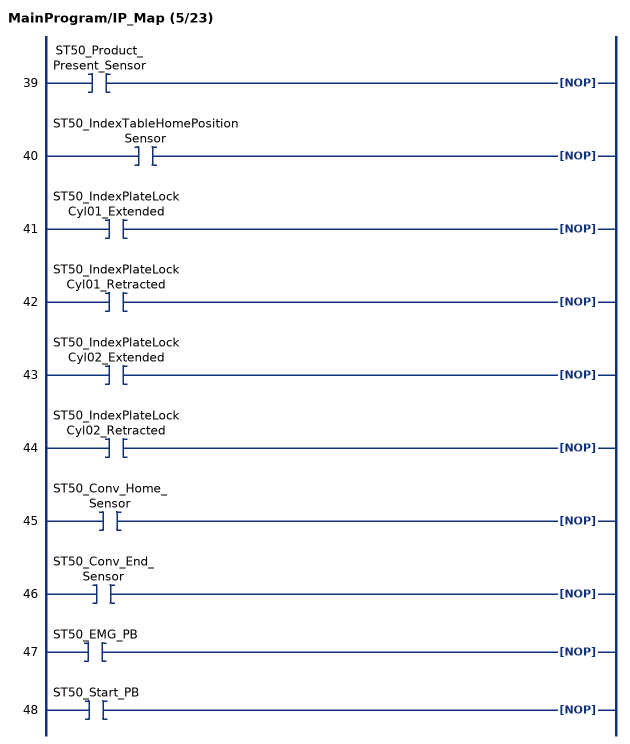
   39: XIC(ST50_Product_Present_Sensor)NOP();
   40: XIC(ST50_IndexTableHomePositionSensor)NOP();
   41: XIC(ST50_IndexPlateLockCyl01_Extended)NOP();
   42: XIC(ST50_IndexPlateLockCyl01_Retracted)NOP();
   43: XIC(ST50_IndexPlateLockCyl02_Extended)NOP();
   44: XIC(ST50_IndexPlateLockCyl02_Retracted)NOP();
   45: XIC(ST50_Conv_Home_Sensor)NOP();
   46: XIC(ST50_Conv_End_Sensor)NOP();
   47: XIC(ST50_EMG_PB)NOP();
   48: XIC(ST50_Start_PB)NOP();
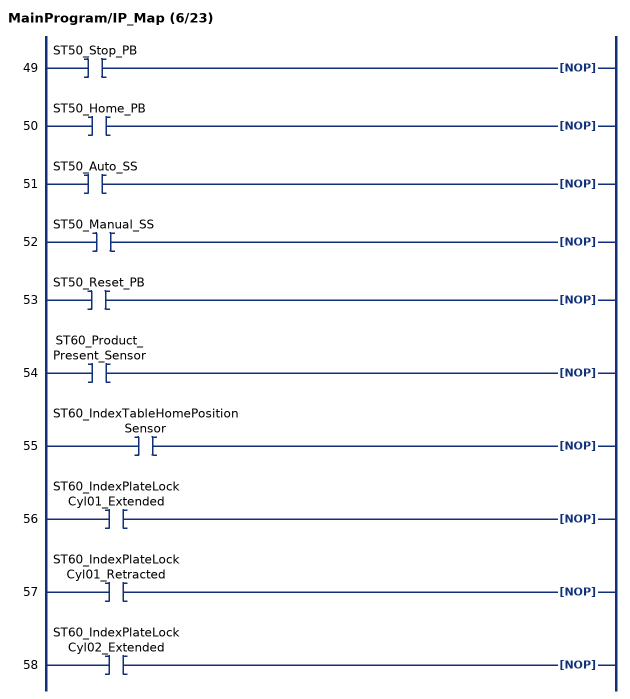
   49: XIC(ST50_Stop_PB)NOP();
   50: XIC(ST50_Home_PB)NOP();
   51: XIC(ST50_Auto_SS)NOP();
   52: XIC(ST50_Manual_SS)NOP();
   53: XIC(ST50_Reset_PB)NOP();
   54: XIC(ST60_Product_Present_Sensor)NOP();
   55: XIC(ST60_IndexTableHomePositionSensor)NOP();
   56: XIC(ST60_IndexPlateLockCyl01_Extended)NOP();
   57: XIC(ST60_IndexPlateLockCyl01_Retracted)NOP();
   58: XIC(ST60_IndexPlateLockCyl02_Extended)NOP();
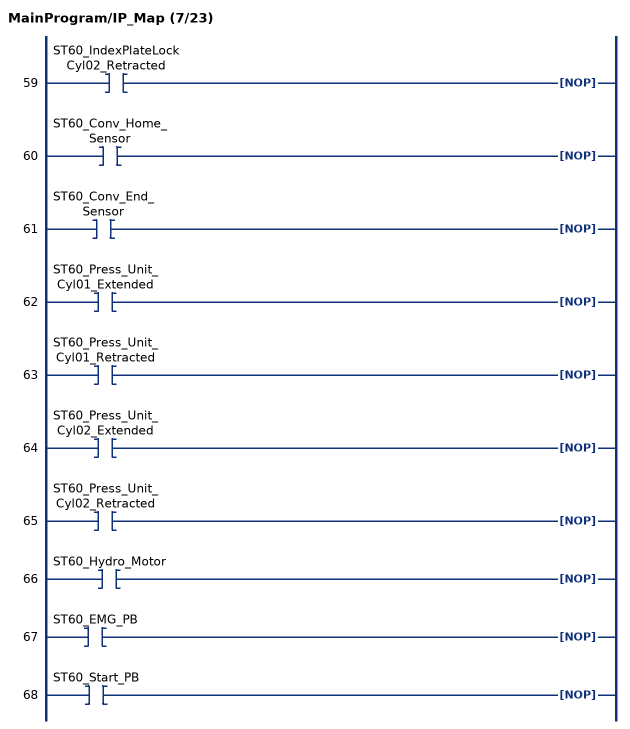
   59: XIC(ST60_IndexPlateLockCyl02_Retracted)NOP();
   60: XIC(ST60_Conv_Home_Sensor)NOP();
   61: XIC(ST60_Conv_End_Sensor)NOP();
   62: XIC(ST60_Press_Unit_Cyl01_Extended)NOP();
   63: XIC(ST60_Press_Unit_Cyl01_Retracted)NOP();
   64: XIC(ST60_Press_Unit_Cyl02_Extended)NOP();
   65: XIC(ST60_Press_Unit_Cyl02_Retracted)NOP();
   66: XIC(ST60_Hydro_Motor)NOP();
   67: XIC(ST60_EMG_PB)NOP();
   68: XIC(ST60_Start_PB)NOP();
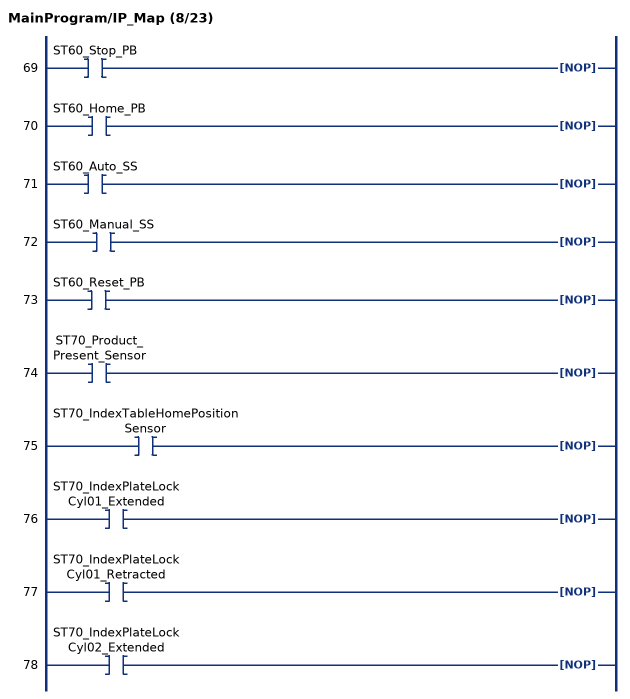
   69: XIC(ST60_Stop_PB)NOP();
   70: XIC(ST60_Home_PB)NOP();
   71: XIC(ST60_Auto_SS)NOP();
   72: XIC(ST60_Manual_SS)NOP();
   73: XIC(ST60_Reset_PB)NOP();
   74: XIC(ST70_Product_Present_Sensor)NOP();
   75: XIC(ST70_IndexTableHomePositionSensor)NOP();
   76: XIC(ST70_IndexPlateLockCyl01_Extended)NOP();
   77: XIC(ST70_IndexPlateLockCyl01_Retracted)NOP();
   78: XIC(ST70_IndexPlateLockCyl02_Extended)NOP();
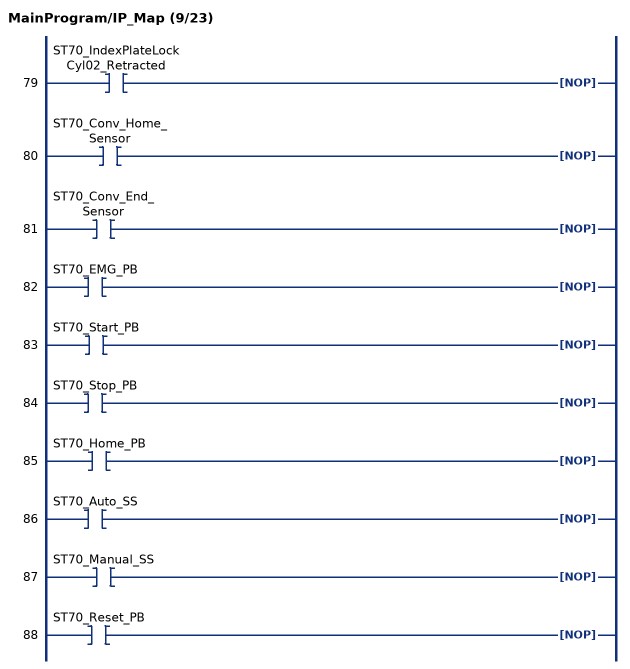
   79: XIC(ST70_IndexPlateLockCyl02_Retracted)NOP();
   80: XIC(ST70_Conv_Home_Sensor)NOP();
   81: XIC(ST70_Conv_End_Sensor)NOP();
   82: XIC(ST70_EMG_PB)NOP();
   83: XIC(ST70_Start_PB)NOP();
   84: XIC(ST70_Stop_PB)NOP();
   85: XIC(ST70_Home_PB)NOP();
   86: XIC(ST70_Auto_SS)NOP();
   87: XIC(ST70_Manual_SS)NOP();
   88: XIC(ST70_Reset_PB)NOP();
